// TwinCAT 3 PLC project Untitled1
// ProgramVersion: 3.1.4023.0
// libraries:
//   Tc2_Standard, * (Beckhoff Automation GmbH)
//   Tc2_System, * (Beckhoff Automation GmbH)
//   Tc3_Module, * (Beckhoff Automation GmbH)
// project tree:
//   / PlcTask.TcTTO
//   POUs/ MAIN.TcPOU

CONFIGURATION Untitled1
    RESOURCE PLC ON TwinCAT3
        TASK PlcTask(INTERVAL := T#10ms, PRIORITY := 20);
        PROGRAM MAIN WITH PlcTask : MAIN;
    END_RESOURCE
END_CONFIGURATION

// ---- POUs/MAIN.TcPOU
PROGRAM MAIN
VAR
	PLCVar AT %MD0 : DWORD;
	PCVar AT %MD1 : DWORD;
	TP_1		: TP;
	TOGGEL: BOOL;
END_VAR

TOGGEL := NOT TOGGEL;
TP_1( IN := TOGGEL, PT := T#4S);
IF (TP_1.Q = 0) THEN
	PLCVar := PLCVar + 1;
	TOGGEL := NOT TOGGEL;
	TP_1( IN := TOGGEL, PT := T#4S);
END_IF

END_PROGRAM
